FUNCTION_BLOCK AIS2_TO_AIS (* Composite FB for convert bidirectional AIS2 to unidirectional AIS *)
  (* Standard: 61499-2; Function: AIS2_BIDIR forwards its incoming (EO1) side out as a plain unidirectional signal via AIS_OUT. AIS_IN publishes its value onto the outgoing (EI1) side of AIS2_BIDIR.; Description: Copyright (c) 2026 HR Agrartechnik GmbH This program and the accompanying materials are made available under the terms of the Eclipse Public License 2.0 which is available at https://www.eclipse.org/legal/epl-2.0/ SPDX-License-Identifier: EPL-2.0 *)
  (* Version 1.0, 2026-09-12, Franz Höpfinger, HR Agrartechnik GmbH, Initial Version - Konvertierungsfamilie vervollstaendigt (analog zu AR2/AB2/AE2). *)
  PACKAGE adapter::conversion::bidirectional;
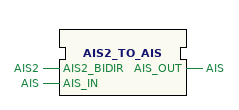
  SOCKETS
    AIS2_BIDIR : adapter::types::bidirectional::AIS2; (* Adapter Input: bidirectional tap, incoming side forwarded to AIS_OUT, outgoing side driven by AIS_IN *)
    AIS_IN : adapter::types::unidirectional::AIS; (* Adapter Input: unidirectional source *)
  END_SOCKETS
  PLUGS
    AIS_OUT : adapter::types::unidirectional::AIS; (* Adapter Output: mirrors AIS2_BIDIR's incoming (indication) side *)
  END_PLUGS
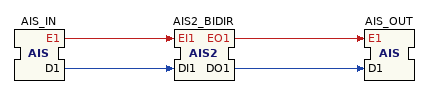
  EVENT_CONNECTIONS
    AIS2_BIDIR.EO1 TO AIS_OUT.E1;
    AIS_IN.E1 TO AIS2_BIDIR.EI1;
  END_CONNECTIONS
  DATA_CONNECTIONS
    AIS2_BIDIR.DO1 TO AIS_OUT.D1;
    AIS_IN.D1 TO AIS2_BIDIR.DI1;
  END_CONNECTIONS
END_FUNCTION_BLOCK
